ABB RobotStudio station: Est_1.rsstn

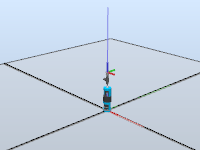
Station Solution14 (saved by RobotStudio 20.1.9056.2)
Layout (positions relative to the parent item):
  - smc_gripper [mechanism] at (0, 0, 0) mm
      TCP smc_gripper at (51.61, 2.43, -191.63) mm, rotated rx 180 ry 0 rz 180 deg
      links: smc_end_effector
  - Frame_1 [frame] at (0, 0, 197) mm
